FUNCTION_BLOCK CNV_MERGE_MDL (* Composite Function Block Type *)
  (* Standard: 61499-2 *)
  (* Version 0.2, 2003-12-05, JHC, Rockwell Automation, Renamed from NEWCOMPFB. *)
  (* Version 0.1, 2002-01-08, JHC, Rockwell Automation, Added DLY FB as example. *)
  (* Version 0.0, 2000-05-27, JHC, Rockwell Automation *)
  PACKAGE fb.rt.Conveyer;
  IMPORT fb.datatype.*;
  IMPORT fb.rt.*;
  IMPORT fb.rt.events.E_PERMIT;
  IMPORT fb.rt.math.FB_AND;
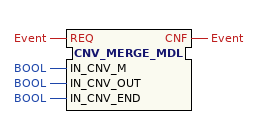
  EVENT_INPUT
    REQ;
  END_EVENT
  EVENT_OUTPUT
    CNF;
  END_EVENT
  VAR_INPUT
    IN_CNV_M : BOOL;
    IN_CNV_OUT : BOOL;
    IN_CNV_END : BOOL;
  END_VAR
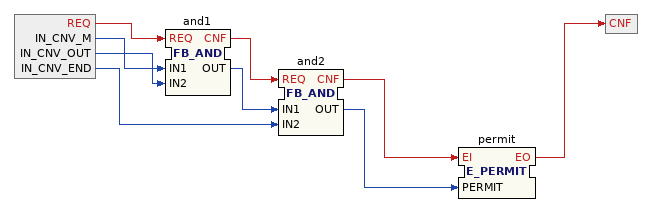
  FBS
    and1 : FB_AND;
    and2 : FB_AND;
    permit : E_PERMIT;
  END_FBS
  EVENT_CONNECTIONS
    and1.CNF TO and2.REQ;
    and2.CNF TO permit.EI;
    permit.EO TO CNF;
    REQ TO and1.REQ;
  END_CONNECTIONS
  DATA_CONNECTIONS
    and1.OUT TO and2.IN1;
    IN_CNV_M TO and1.IN1;
    IN_CNV_OUT TO and1.IN2;
    IN_CNV_END TO and2.IN2;
    and2.OUT TO permit.PERMIT;
  END_CONNECTIONS
END_FUNCTION_BLOCK
